Fanuc TP program (LS listing): SHIP.LS

/PROG  SHIP
/ATTR
OWNER		= MNEDITOR;
COMMENT		= "";
PROG_SIZE	= 536;
CREATE		= DATE 20-10-13  TIME 22:16:58;
MODIFIED	= DATE 21-02-04  TIME 12:10:36;
FILE_NAME	= ZERO;
VERSION		= 0;
LINE_COUNT	= 1;
MEMORY_SIZE	= 904;
PROTECT		= READ_WRITE;
TCD:  STACK_SIZE	= 0,
      TASK_PRIORITY	= 50,
      TIME_SLICE	= 0,
      BUSY_LAMP_OFF	= 0,
      ABORT_REQUEST	= 0,
      PAUSE_REQUEST	= 0;
DEFAULT_GROUP	= 1,*,*,*,*;
CONTROL_CODE	= 00000000 00000000;
/APPL
/APPL

AUTO_SINGULARITY_HEADER;
  ENABLE_SINGULARITY_AVOIDANCE   : TRUE;

  AUTOZONE_INTERFERENCE_AVOID;
    AUTOZONE_ENABLED         : FALSE;
    AUTOZONE_SCHEDULE_NUMBER : 1;
/MN
   1:J P[1] 100% FINE    ;
/POS
P[1]{
   GP1:
	UF : 0, UT : 1,
	J1=     1.211 deg,	J2=   -18.835 deg,	J3=   -61.320 deg,
	J4=    90.857 deg,	J5=    92.250 deg,	J6=     -.000 deg
};
/END
